FUNCTION_BLOCK FB_System_HOWW_Ablaufsteuerung
VAR_IN_OUT
	Zustand					: ST_System_HOWW_Zustand;
	Stellwert				: ST_System_HOWW_Stellwert;
	Steuerung				: ST_System_HOWW_Steuerung;
END_VAR
VAR_INPUT
	Zustand_Regelventil		: ST_RV_Zustand;
	Zustand_Pumpe			: ST_PU_Zustand;
END_VAR
VAR_OUTPUT
END_VAR
VAR
END_VAR

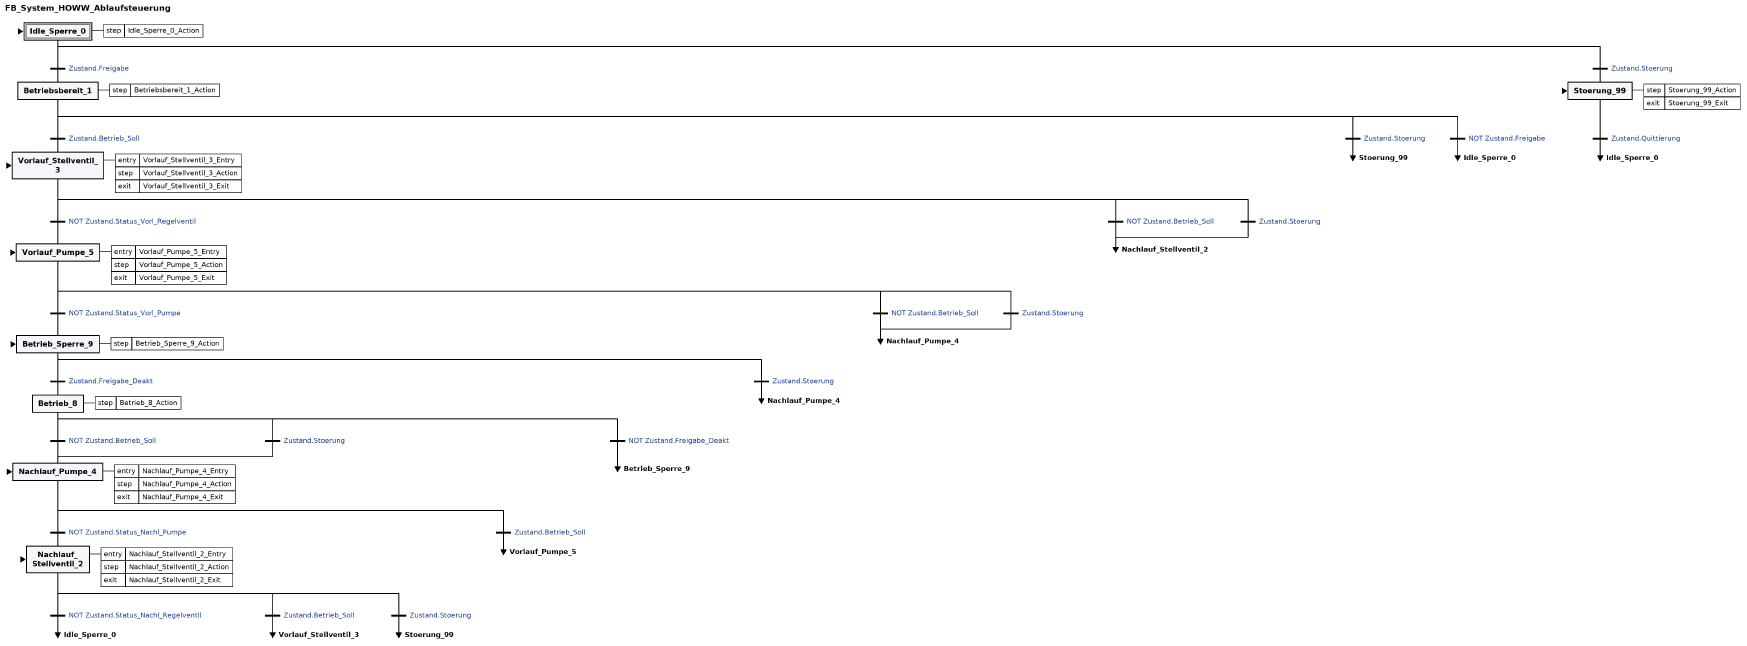
INITIAL_STEP Idle_Sperre_0:
    Idle_Sperre_0_Action(N);  // step action
END_STEP
TRANSITION FROM Idle_Sperre_0 TO Betriebsbereit_1
    := Zustand.Freigabe;
END_TRANSITION
TRANSITION FROM Idle_Sperre_0 TO Stoerung_99
    := Zustand.Stoerung;
END_TRANSITION
STEP Stoerung_99:
    Stoerung_99_Action(N);  // step action
    Stoerung_99_Exit(P0);  // exit action
END_STEP
TRANSITION FROM Stoerung_99 TO Idle_Sperre_0
    := Zustand.Quittierung;
END_TRANSITION
STEP Betriebsbereit_1:
    Betriebsbereit_1_Action(N);  // step action
END_STEP
TRANSITION FROM Betriebsbereit_1 TO Vorlauf_Stellventil_3
    := Zustand.Betrieb_Soll;
END_TRANSITION
TRANSITION FROM Betriebsbereit_1 TO Stoerung_99
    := Zustand.Stoerung;
END_TRANSITION
TRANSITION FROM Betriebsbereit_1 TO Idle_Sperre_0
    := NOT Zustand.Freigabe;
END_TRANSITION
STEP Vorlauf_Stellventil_3:
    Vorlauf_Stellventil_3_Entry(P1);  // entry action
    Vorlauf_Stellventil_3_Action(N);  // step action
    Vorlauf_Stellventil_3_Exit(P0);  // exit action
END_STEP
TRANSITION FROM Vorlauf_Stellventil_3 TO Vorlauf_Pumpe_5
    := NOT Zustand.Status_Vorl_Regelventil;
END_TRANSITION
TRANSITION FROM Vorlauf_Stellventil_3 TO Nachlauf_Stellventil_2
    := NOT Zustand.Betrieb_Soll;
END_TRANSITION
TRANSITION FROM Vorlauf_Stellventil_3 TO Nachlauf_Stellventil_2
    := Zustand.Stoerung;
END_TRANSITION
STEP Vorlauf_Pumpe_5:
    Vorlauf_Pumpe_5_Entry(P1);  // entry action
    Vorlauf_Pumpe_5_Action(N);  // step action
    Vorlauf_Pumpe_5_Exit(P0);  // exit action
END_STEP
TRANSITION FROM Vorlauf_Pumpe_5 TO Betrieb_Sperre_9
    := NOT Zustand.Status_Vorl_Pumpe;
END_TRANSITION
TRANSITION FROM Vorlauf_Pumpe_5 TO Nachlauf_Pumpe_4
    := NOT Zustand.Betrieb_Soll;
END_TRANSITION
TRANSITION FROM Vorlauf_Pumpe_5 TO Nachlauf_Pumpe_4
    := Zustand.Stoerung;
END_TRANSITION
STEP Betrieb_Sperre_9:
    Betrieb_Sperre_9_Action(N);  // step action
END_STEP
TRANSITION FROM Betrieb_Sperre_9 TO Betrieb_8
    := Zustand.Freigabe_Deakt;
END_TRANSITION
TRANSITION FROM Betrieb_Sperre_9 TO Nachlauf_Pumpe_4
    := Zustand.Stoerung;
END_TRANSITION
STEP Betrieb_8:
    Betrieb_8_Action(N);  // step action
END_STEP
TRANSITION FROM Betrieb_8 TO Nachlauf_Pumpe_4
    := NOT Zustand.Betrieb_Soll;
END_TRANSITION
TRANSITION FROM Betrieb_8 TO Nachlauf_Pumpe_4
    := Zustand.Stoerung;
END_TRANSITION
TRANSITION FROM Betrieb_8 TO Betrieb_Sperre_9
    := NOT Zustand.Freigabe_Deakt;
END_TRANSITION
STEP Nachlauf_Pumpe_4:
    Nachlauf_Pumpe_4_Entry(P1);  // entry action
    Nachlauf_Pumpe_4_Action(N);  // step action
    Nachlauf_Pumpe_4_Exit(P0);  // exit action
END_STEP
TRANSITION FROM Nachlauf_Pumpe_4 TO Nachlauf_Stellventil_2
    := NOT Zustand.Status_Nachl_Pumpe;
END_TRANSITION
TRANSITION FROM Nachlauf_Pumpe_4 TO Vorlauf_Pumpe_5
    := Zustand.Betrieb_Soll;
END_TRANSITION
STEP Nachlauf_Stellventil_2:
    Nachlauf_Stellventil_2_Entry(P1);  // entry action
    Nachlauf_Stellventil_2_Action(N);  // step action
    Nachlauf_Stellventil_2_Exit(P0);  // exit action
END_STEP
TRANSITION FROM Nachlauf_Stellventil_2 TO Idle_Sperre_0
    := NOT Zustand.Status_Nachl_Regelventil;
END_TRANSITION
TRANSITION FROM Nachlauf_Stellventil_2 TO Vorlauf_Stellventil_3
    := Zustand.Betrieb_Soll;
END_TRANSITION
TRANSITION FROM Nachlauf_Stellventil_2 TO Stoerung_99
    := Zustand.Stoerung;
END_TRANSITION

ACTION Betrieb_8_Action:
(* Stellwert setzen *)
Stellwert.Anford_Stellventil	:= TRUE;
Stellwert.Anford_Pumpe	:= TRUE;
Stellwert.Freigabe_Anlage	:= TRUE;

(* Zustand setzen *)
Zustand.Status				:= E_System_HO_Zustand_Status_Betrieb;
END_ACTION

ACTION Betrieb_Sperre_9_Action:
(* Stellwert setzen *)
Stellwert.Anford_Stellventil	:= TRUE;
Stellwert.Anford_Pumpe	:= TRUE;
Stellwert.Freigabe_Anlage	:= TRUE;

(* Zustand setzen *)
Zustand.Status				:= E_System_HO_Zustand_Status_Betrieb_Sperre;
END_ACTION

ACTION Betriebsbereit_1_Action:
(* Stellwert setzen *)
Stellwert.Anford_Stellventil	:= FALSE;
Stellwert.Anford_Pumpe	:= FALSE;
Stellwert.Freigabe_Anlage	:= FALSE;

(* Zustand setzen *)
Zustand.Status			:= E_System_HO_Zustand_Status_Betriebsbereit;
END_ACTION

ACTION Idle_Sperre_0_Action:
(* Stellwert setzen *)
Stellwert.Anford_Stellventil	:= FALSE;
Stellwert.Anford_Pumpe	:= FALSE;
Stellwert.Freigabe_Anlage	:= FALSE;

(* Zustand setzen *)
Zustand.Status			:= E_System_HO_Zustand_Status_Idle_Sperre;

(* Quittierungszustand auf False setzen, damit das System bei einer erneuten Störung nicht direkt wieder angeschaltet wird *)
Steuerung.Quittierung	:= FALSE;
END_ACTION

ACTION Nachlauf_Pumpe_4_Action:
(* Stellwert setzen *)
Stellwert.Anford_Stellventil	:= TRUE;
Stellwert.Anford_Pumpe	:= FALSE;
Stellwert.Freigabe_Anlage	:= FALSE;

(* Zustand setzen *)
Zustand.Status				:= E_System_HO_Zustand_Status_Nachl_Pumpe;
Zustand.Status_Nachl_Pumpe	:= Zustand_Pumpe.Betrieb OR Zustand_Pumpe.Status_Nachl;
END_ACTION

ACTION Nachlauf_Pumpe_4_Entry:
Zustand.Status_Nachl_Pumpe	:= TRUE;
END_ACTION

ACTION Nachlauf_Pumpe_4_Exit:
Zustand.Status_Nachl_Pumpe	:= FALSE;
END_ACTION

ACTION Nachlauf_Stellventil_2_Action:
(* Stellwert setzen *)
Stellwert.Anford_Stellventil	:= FALSE;
Stellwert.Anford_Pumpe	:= FALSE;
Stellwert.Freigabe_Anlage	:= FALSE;

(* Zustand setzen *)
Zustand.Status				:= E_System_HO_Zustand_Status_Nachl_Regelventil;
Zustand.Status_Nachl_Regelventil	:= Zustand_Regelventil.Betrieb OR Zustand_Regelventil.Status_Nachl;
END_ACTION

ACTION Nachlauf_Stellventil_2_Entry:
Zustand.Status_Nachl_Regelventil	:= TRUE;
END_ACTION

ACTION Nachlauf_Stellventil_2_Exit:
Zustand.Status_Nachl_Regelventil	:= FALSE;
END_ACTION

ACTION Stoerung_99_Action:
(* Stellwert setzen *)
Stellwert.Anford_Stellventil	:= FALSE;
Stellwert.Anford_Pumpe	:= FALSE;
Stellwert.Freigabe_Anlage	:= FALSE;

(* Zustand setzen *)
Zustand.Stoerung			:= TRUE;
Zustand.Status			:= E_System_HO_Zustand_Status_Stoerung;
END_ACTION

ACTION Stoerung_99_Exit:
Zustand.Stoerung	:= FALSE;
END_ACTION

ACTION Vorlauf_Pumpe_5_Action:
(* Stellwert setzen *)
Stellwert.Anford_Stellventil	:= TRUE;
Stellwert.Anford_Pumpe	:= TRUE;
Stellwert.Freigabe_Anlage	:= FALSE;

(* Zustand setzen *)
Zustand.Status				:= E_System_HO_Zustand_Status_Vorl_Pumpe;
Zustand.Status_Vorl_Pumpe	:= NOT(Zustand_Pumpe.Betrieb AND NOT Zustand_Pumpe.Status_Vorl);
END_ACTION

ACTION Vorlauf_Pumpe_5_Entry:
Zustand.Status_Vorl_Pumpe	:= TRUE;
END_ACTION

ACTION Vorlauf_Pumpe_5_Exit:
Zustand.Status_Vorl_Pumpe	:= FALSE;
END_ACTION

ACTION Vorlauf_Stellventil_3_Action:
(* Stellwert setzen *)
Stellwert.Anford_Stellventil	:= TRUE;
Stellwert.Anford_Pumpe	:= FALSE;
Stellwert.Freigabe_Anlage	:= FALSE;

(* Zustand setzen *)
Zustand.Status				:= E_System_HO_Zustand_Status_Vorl_Regelventil;
Zustand.Status_Vorl_Regelventil	:= NOT(Zustand_Regelventil.Betrieb AND NOT Zustand_Regelventil.Status_Vorl);
END_ACTION

ACTION Vorlauf_Stellventil_3_Entry:
Zustand.Status_Vorl_Regelventil	:= TRUE;
END_ACTION

ACTION Vorlauf_Stellventil_3_Exit:
Zustand.Status_Vorl_Regelventil	:= FALSE;
END_ACTION

END_FUNCTION_BLOCK

(* stored: Version 1.1.0.1, ProductVersion 3.1.4024.9
   POU FB_System_HOWW_Ablaufsteuerung: Id {8f23c97a-b3b8-4e27-9df4-4c7e534922d9}, SpecialFunc None
   Action Betrieb_8_Action: Id {9d77cc8c-409b-45ee-99c7-69dff9cf2670}
   Action Betrieb_Sperre_9_Action: Id {d49b045f-a667-4324-ada7-2ba1b25926a2}
   Action Betriebsbereit_1_Action: Id {bae0b0fe-8631-499f-8d78-9769416ad0ee}
   Action Idle_Sperre_0_Action: Id {96d14bd7-5901-4741-908d-22458053390c}
   Action Nachlauf_Pumpe_4_Action: Id {3ab130d2-6a76-41b3-9e86-0f5b370ede99}
   Action Nachlauf_Pumpe_4_Entry: Id {d837d7ef-663c-4f66-984a-f1814ae17117}
   Action Nachlauf_Pumpe_4_Exit: Id {1a2f62f2-f67b-48e0-b3e5-3a680fdeb577}
   Action Nachlauf_Stellventil_2_Action: Id {b98248f3-c70d-419a-a198-0ab810dc5d4e}
   Action Nachlauf_Stellventil_2_Entry: Id {73f1c917-a826-415e-a1c5-9b69b2bea454}
   Action Nachlauf_Stellventil_2_Exit: Id {72fe580f-37e4-4956-a5b1-433df362d1e5}
   Action Stoerung_99_Action: Id {a1e17fbd-58c4-48e2-b327-8d31e1a4583f}
   Action Stoerung_99_Exit: Id {c68d1d43-b855-4c1c-a93b-4799c9a0d78f}
   Action Vorlauf_Pumpe_5_Action: Id {3d6cef59-11a7-46e2-896f-525c7e542c56}
   Action Vorlauf_Pumpe_5_Entry: Id {24eb15b0-6ab3-429e-8589-624e30cea0f0}
   Action Vorlauf_Pumpe_5_Exit: Id {6fa5d407-9878-4cfe-b5c2-2a9997d34a7c}
   Action Vorlauf_Stellventil_3_Action: Id {0c705f67-9f80-49be-8566-110829a81262}
   Action Vorlauf_Stellventil_3_Entry: Id {e48cb84f-f302-4c65-9097-d99be157773b}
   Action Vorlauf_Stellventil_3_Exit: Id {53d05c0a-be20-4bd1-8dfa-81de4b24745a} *)
